// TIA Portal V20 export
DATA_BLOCK "CurrGlob"   // DB3
TITLE = Dati di posizione in coordinate assolute
{ S7_Optimized_Access := 'TRUE' }
// Ottiene la passizione assoluta degli assi
// stored: MemoryReserve 100
   VAR
      Pos : "Position";
   END_VAR
BEGIN
END_DATA_BLOCK
